VAR_GLOBAL
	(*======================= Analog Stacker crane* =======================*)
	RBGEndlageMitte	:	BOOL;
	RBGEndlageLinks	:	BOOL;
	RBGEndlageRechts :	BOOL;
	RBGIstwertX	:	WORD;
	RBGIstwertZ	:	WORD;
	RBGGabelLinks	:	BOOL;
	RBGGabelRechts	:	BOOL;
	RBGSollwertX	:	WORD;
	RBGSollwertZ	:	WORD;
	
(*======================= Simulation* =======================*)
	RBGStartMove	:	BOOL;
	RBGStartForkLeftMove	:	BOOL;
	RBGStartForkRightMove	:	BOOL;
	RBGStartForkMiddleMove	:	BOOL;
	InUnloadingAnalog	:	BOOL;
	RBGSollwertXSimu	:	REAL;
	RBGSollwertZSimu	:	REAL;
	instStackerCraneAnalog	:	FB_StackerCrane_Analog;
	processStepsAnalogStackerCrane	: StackerCraneSteps;
	
(*======================= Numerical Stacker crane* =======================*)	
	DigitalStackerCraneEndlageMitte	:	BOOL;
	DigitalStackerCraneEndlageLinks	:	BOOL;
	DigitalStackerCraneEndlageRechts :	BOOL;
	DigitalStackerCraneGabelLinks	:	BOOL;
	DigitalStackerCraneGabelRechts	:	BOOL;
	DigitalStackerCraneLiftGabel	:	BOOL;
	DigitalStackerCraneXAxisIsMoving	:	BOOL;
	DigitalStackerCraneZAxisIsMoving	:	BOOL;
	DigitalStackerCraneTargetPos	:	WORD;
	
	(*======================= Simulation* =======================*)
	DigtalStackerCraneStartMove	:	BOOL;
	DigtalStackerCraneStartForkLeftMove	:	BOOL;
	DigtalStackerCraneStartForkRightMove	:	BOOL;
	DigtalStackerCraneStartForkMiddleMove	:	BOOL;
	DigitalStackerCraneStartLiftFork	:	BOOL;
	InUnloadingNumerical	:	BOOL;
	Lifting	:	BOOL;
	Lowering	:	BOOL;
	DigitalTargetPosSimu	:	WORD := 7;
	instStackerCraneNumerical	:	FB_StackerCrane_Numerical;
	processStepsNumericalStackerCrane	: StackerCraneSteps;
END_VAR

(* stored: Version 1.1.0.1
   GVL Warehouse: Id {77d69743-90e2-4276-a87d-95431fe3fc7c} *)
